Fanuc KAREL source: ka00130.KL

-- PROVISIONAL review KL for V770-1; original PC SHA256 4756d8ee6fcec615ff6416c914a2b4f27a621c9aa8823b8d8e6a3410a454eaac
-- Incomplete behavior may be omitted. Consult companion uncertainty JSON. Do not deploy.
PROGRAM KA00130
%NOLOCKGROUP
-- UNRESOLVED_DECL SRC type=002018
-- UNRESOLVED_DECL DST type=00001c
BEGIN
  -- UNRESOLVED_PC offsets 5-19; opcodes 2E,22,9D,33,B2
  -- UNRESOLVED_PC offsets 24-39; opcodes 22,9D,33,B1,23
  -- UNRESOLVED_PC offsets 44-48; opcodes 7F
END KA00130
